// TIA Portal project "DALU-Projekt_HMI_V19" (V19)

(* hardware
DEVICE "SIMATIC 1200-Station_3"  S71200.Device
   slot 0: "S7-1200 Baugruppenträger"  Rack  V1.0
   slot 1: "Target_3"  CPU 1214C DC/DC/DC  6ES7 214-1AE30-0XB0  V2.2
   slot 101: "Target 3 CM 1243-2"  CM 1243-2  3RK7243-2AA30-0XB0  V1.0
   slot 102: "Target 3 CM 1243-5"  CM 1243-5  6GK7 243-5DX30-0XE0  V1.0
DEVICE "ASi-3-S9 (4DI)"  AS-i slave
   slot 0: "-"  Rail
   slot 1: "ASi-3-S9 (4DI)"  AS-i Standard Slave  AS-i Standard Slave Universal
      slot 1: "ASi-3-S9 (4DI) [AS-i Slave (D)]"  AS-i Address-Module
      slot 2: "ASi-3-S9 (4DI) [AS-i Slave (A)]"  AS-i Address-Module
      slot 3: "ASi-3-S9 (4DI) [AS-i Slave (T)]"  AS-i Address-Module
DEVICE "ASi-3-S5 (2AI)"  AS-i slave
   slot 0: "-"  Rail
   slot 1: "ASi-3-S5 (2AI)"  AS-i K60, 2AI-C  3RK1 207-1BQ40-0AA3
      slot 1: "ASi-3-S5 (2AI) [AS-i Slave (D)]"  AS-i Address-Module
      slot 2: "ASi-3-S5 (2AI) [AS-i Slave (A)]"  AS-i Address-Module
      slot 3: "ASi-3-S5 (2AI) [AS-i Slave (T)]"  AS-i Address-Module
DEVICE "ASi-3-S1 (4DI/4DO)"  AS-i slave
   slot 0: "-"  Rail
   slot 1: "ASi-3-S1 (4DI/4DO)"  AS-i 3SB3, 4DI/4DO  3SF5 500-0BC
      slot 1: "ASi-3-S1 (4DI/4DO) [AS-i Slave (D)]"  AS-i Address-Module
      slot 2: "ASi-3-S1 (4DI/4DO) [AS-i Slave (A)]"  AS-i Address-Module
      slot 3: "ASi-3-S1 (4DI/4DO) [AS-i Slave (T)]"  AS-i Address-Module
DEVICE "ASi-3-S7 (2DI,2PO)"  AS-i slave
   slot 0: "-"  Rail
   slot 1: "ASi-3-S7 (2DI,2PO)"  AS-i Standard Slave  AS-i Standard Slave Universal
      slot 1: "ASi-3-S7 (2DI,2PO) [AS-i Slave (D)]"  AS-i Address-Module
      slot 2: "ASi-3-S7 (2DI,2PO) [AS-i Slave (A)]"  AS-i Address-Module
      slot 3: "ASi-3-S7 (2DI,2PO) [AS-i Slave (T)]"  AS-i Address-Module
DEVICE "ASi-3-S3 (2AI)"  AS-i slave
   slot 0: "-"  Rail
   slot 1: "ASi-3-S3 (2AI)"  AS-i K60, 2AI-V  3RK1 207-2BQ40-0AA3
      slot 1: "ASi-3-S3 (2AI) [AS-i Slave (D)]"  AS-i Address-Module
      slot 2: "ASi-3-S3 (2AI) [AS-i Slave (A)]"  AS-i Address-Module
      slot 3: "ASi-3-S3 (2AI) [AS-i Slave (T)]"  AS-i Address-Module
DEVICE "ASi-3-S8 (3DI/1DO)"  AS-i slave
   slot 0: "-"  Rail
   slot 1: "ASi-3-S8 (3DI/1DO)"  AS-i Standard Slave  AS-i Standard Slave Universal
      slot 1: "ASi-3-S8 (3DI/1DO) [AS-i Slave (D)]"  AS-i Address-Module
      slot 2: "ASi-3-S8 (3DI/1DO) [AS-i Slave (A)]"  AS-i Address-Module
      slot 3: "ASi-3-S8 (3DI/1DO) [AS-i Slave (T)]"  AS-i Address-Module
DEVICE "DP_3_S1"  GSD.Device
   slot 0: "Baugruppenträger"  Rail
   slot 0: "DP_3_Simodrive"  6FX2001-5xPxx  4.2
DEVICE "ASi-3-S2 (2AO)"  AS-i slave
   slot 0: "-"  Rail
   slot 1: "ASi-3-S2 (2AO)"  AS-i K60, 2AO-V  3RK1 107-2BQ40-0AA3
      slot 1: "ASi-3-S2 (2AO) [AS-i Slave (D)]"  AS-i Address-Module
      slot 2: "ASi-3-S2 (2AO) [AS-i Slave (A)]"  AS-i Address-Module
      slot 3: "ASi-3-S2 (2AO) [AS-i Slave (T)]"  AS-i Address-Module
DEVICE "ASi-3-S4 (4DI/4DO)"  AS-i slave
   slot 0: "-"  Rail
   slot 1: "ASi-3-S4 (4DI/4DO)"  AS-i K60, 4DI/4DO  3RK1 400-1DQ01-0AA3
      slot 1: "ASi-3-S4 (4DI/4DO) [AS-i Slave (D)]"  AS-i Address-Module
      slot 2: "ASi-3-S4 (4DI/4DO) [AS-i Slave (A)]"  AS-i Address-Module
      slot 3: "ASi-3-S4 (4DI/4DO) [AS-i Slave (T)]"  AS-i Address-Module
DEVICE "ASi-3-S6 (4DI)"  AS-i slave
   slot 0: "-"  Rail
   slot 1: "ASi-3-S6 (4DI)"  AS-i K45, 4DI  3RK1 200-0CQ20-0AA3
      slot 1: "ASi-3-S6 (4DI) [AS-i Slave (D)]"  AS-i Address-Module
      slot 2: "ASi-3-S6 (4DI) [AS-i Slave (A)]"  AS-i Address-Module
      slot 3: "ASi-3-S6 (4DI) [AS-i Slave (T)]"  AS-i Address-Module
DEVICE "SIMATIC 1200-Station_4"  S71200.Device
   slot 0: "S7-1200 Baugruppenträger"  Rack  V1.0
   slot 1: "Target_4"  CPU 1214C DC/DC/DC  6ES7 214-1AE30-0XB0  V2.2
   slot 101: "Target 4 CM 1243-2"  CM 1243-2  3RK7243-2AA30-0XB0  V1.0
   slot 102: "Target 4 CM 1243-5"  CM 1243-5  6GK7 243-5DX30-0XE0  V1.0
DEVICE "ASi-4-S9 (4DI)"  AS-i slave
   slot 0: "-"  Rail
   slot 1: "ASi-4-S9 (4DI)"  AS-i Standard Slave  AS-i Standard Slave Universal
      slot 1: "ASi-4-S9 (4DI) [AS-i Slave (D)]"  AS-i Address-Module
      slot 2: "ASi-4-S9 (4DI) [AS-i Slave (A)]"  AS-i Address-Module
      slot 3: "ASi-4-S9 (4DI) [AS-i Slave (T)]"  AS-i Address-Module
DEVICE "ASi-4-S5 (2AI)"  AS-i slave
   slot 0: "-"  Rail
   slot 1: "ASi-4-S5 (2AI)"  AS-i K60, 2AI-C  3RK1 207-1BQ40-0AA3
      slot 1: "ASi-4-S5 (2AI) [AS-i Slave (D)]"  AS-i Address-Module
      slot 2: "ASi-4-S5 (2AI) [AS-i Slave (A)]"  AS-i Address-Module
      slot 3: "ASi-4-S5 (2AI) [AS-i Slave (T)]"  AS-i Address-Module
DEVICE "ASi-4-S1 (4DI/4DO)"  AS-i slave
   slot 0: "-"  Rail
   slot 1: "ASi-4-S1 (4DI/4DO)"  AS-i 3SB3, 4DI/4DO  3SF5 500-0BC
      slot 1: "ASi-4-S1 (4DI/4DO) [AS-i Slave (D)]"  AS-i Address-Module
      slot 2: "ASi-4-S1 (4DI/4DO) [AS-i Slave (A)]"  AS-i Address-Module
      slot 3: "ASi-4-S1 (4DI/4DO) [AS-i Slave (T)]"  AS-i Address-Module
DEVICE "ASi-4-S7 (2DI,2PO)"  AS-i slave
   slot 0: "-"  Rail
   slot 1: "ASi-4-S7 (2DI,2PO)"  AS-i Standard Slave  AS-i Standard Slave Universal
      slot 1: "ASi-4-S7 (2DI,2PO) [AS-i Slave (D)]"  AS-i Address-Module
      slot 2: "ASi-4-S7 (2DI,2PO) [AS-i Slave (A)]"  AS-i Address-Module
      slot 3: "ASi-4-S7 (2DI,2PO) [AS-i Slave (T)]"  AS-i Address-Module
DEVICE "ASi-4-S3 (2AI)"  AS-i slave
   slot 0: "-"  Rail
   slot 1: "ASi-4-S3 (2AI)"  AS-i K60, 2AI-V  3RK1 207-2BQ40-0AA3
      slot 1: "ASi-4-S3 (2AI) [AS-i Slave (D)]"  AS-i Address-Module
      slot 2: "ASi-4-S3 (2AI) [AS-i Slave (A)]"  AS-i Address-Module
      slot 3: "ASi-4-S3 (2AI) [AS-i Slave (T)]"  AS-i Address-Module
DEVICE "ASi-4-S8 (3DI/1DO)"  AS-i slave
   slot 0: "-"  Rail
   slot 1: "ASi-4-S8 (3DI/1DO)"  AS-i Standard Slave  AS-i Standard Slave Universal
      slot 1: "ASi-4-S8 (3DI/1DO) [AS-i Slave (D)]"  AS-i Address-Module
      slot 2: "ASi-4-S8 (3DI/1DO) [AS-i Slave (A)]"  AS-i Address-Module
      slot 3: "ASi-4-S8 (3DI/1DO) [AS-i Slave (T)]"  AS-i Address-Module
DEVICE "DP_4_S1"  GSD.Device
   slot 0: "Baugruppenträger"  Rail
   slot 0: "DP_4_Simodrive"  6FX2001-5xPxx  4.2
DEVICE "ASi-4-S2 (2AO)"  AS-i slave
   slot 0: "-"  Rail
   slot 1: "ASi-4-S2 (2AO)"  AS-i K60, 2AO-V  3RK1 107-2BQ40-0AA3
      slot 1: "ASi-4-S2 (2AO) [AS-i Slave (D)]"  AS-i Address-Module
      slot 2: "ASi-4-S2 (2AO) [AS-i Slave (A)]"  AS-i Address-Module
      slot 3: "ASi-4-S2 (2AO) [AS-i Slave (T)]"  AS-i Address-Module
DEVICE "ASi-4-S4 (4DI/4DO)"  AS-i slave
   slot 0: "-"  Rail
   slot 1: "ASi-4-S4 (4DI/4DO)"  AS-i K60, 4DI/4DO  3RK1 400-1DQ01-0AA3
      slot 1: "ASi-4-S4 (4DI/4DO) [AS-i Slave (D)]"  AS-i Address-Module
      slot 2: "ASi-4-S4 (4DI/4DO) [AS-i Slave (A)]"  AS-i Address-Module
      slot 3: "ASi-4-S4 (4DI/4DO) [AS-i Slave (T)]"  AS-i Address-Module
DEVICE "ASi-4-S6 (4DI)"  AS-i slave
   slot 0: "-"  Rail
   slot 1: "ASi-4-S6 (4DI)"  AS-i K45, 4DI  3RK1 200-0CQ20-0AA3
      slot 1: "ASi-4-S6 (4DI) [AS-i Slave (D)]"  AS-i Address-Module
      slot 2: "ASi-4-S6 (4DI) [AS-i Slave (A)]"  AS-i Address-Module
      slot 3: "ASi-4-S6 (4DI) [AS-i Slave (T)]"  AS-i Address-Module
DEVICE "SIMATIC 1200-Station_5"  S71200.Device
   slot 0: "S7-1200 Baugruppenträger"  Rack  V1.0
   slot 1: "Target_5"  CPU 1214C DC/DC/DC  6ES7 214-1AE30-0XB0  V2.2
   slot 101: "Target 5 CM 1243-2"  CM 1243-2  3RK7243-2AA30-0XB0  V1.0
   slot 102: "Target 5 CM 1243-5"  CM 1243-5  6GK7 243-5DX30-0XE0  V1.0
DEVICE "ASi-5-S9 (4DI)"  AS-i slave
   slot 0: "-"  Rail
   slot 1: "ASi-5-S9 (4DI)"  AS-i Standard Slave  AS-i Standard Slave Universal
      slot 1: "ASi-5-S9 (4DI) [AS-i Slave (D)]"  AS-i Address-Module
      slot 2: "ASi-5-S9 (4DI) [AS-i Slave (A)]"  AS-i Address-Module
      slot 3: "ASi-5-S9 (4DI) [AS-i Slave (T)]"  AS-i Address-Module
DEVICE "ASi-5-S5 (2AI)"  AS-i slave
   slot 0: "-"  Rail
   slot 1: "ASi-5-S5 (2AI)"  AS-i K60, 2AI-C  3RK1 207-1BQ40-0AA3
      slot 1: "ASi-5-S5 (2AI) [AS-i Slave (D)]"  AS-i Address-Module
      slot 2: "ASi-5-S5 (2AI) [AS-i Slave (A)]"  AS-i Address-Module
      slot 3: "ASi-5-S5 (2AI) [AS-i Slave (T)]"  AS-i Address-Module
DEVICE "ASi-5-S3 (2AI)"  AS-i slave
   slot 0: "-"  Rail
   slot 1: "ASi-5-S3 (2AI)"  AS-i K60, 2AI-V  3RK1 207-2BQ40-0AA3
      slot 1: "ASi-5-S3 (2AI) [AS-i Slave (D)]"  AS-i Address-Module
      slot 2: "ASi-5-S3 (2AI) [AS-i Slave (A)]"  AS-i Address-Module
      slot 3: "ASi-5-S3 (2AI) [AS-i Slave (T)]"  AS-i Address-Module
DEVICE "ASi-5-S7 (2DI,2PO)"  AS-i slave
   slot 0: "-"  Rail
   slot 1: "ASi-5-S7 (2DI,2PO)"  AS-i Standard Slave  AS-i Standard Slave Universal
      slot 1: "ASi-5-S7 (2DI,2PO) [AS-i Slave (D)]"  AS-i Address-Module
      slot 2: "ASi-5-S7 (2DI,2PO) [AS-i Slave (A)]"  AS-i Address-Module
      slot 3: "ASi-5-S7 (2DI,2PO) [AS-i Slave (T)]"  AS-i Address-Module
DEVICE "ASi-5-S2 (2AO)"  AS-i slave
   slot 0: "-"  Rail
   slot 1: "ASi-5-S2 (2AO)"  AS-i K60, 2AO-V  3RK1 107-2BQ40-0AA3
      slot 1: "ASi-5-S2 (2AO) [AS-i Slave (D)]"  AS-i Address-Module
      slot 2: "ASi-5-S2 (2AO) [AS-i Slave (A)]"  AS-i Address-Module
      slot 3: "ASi-5-S2 (2AO) [AS-i Slave (T)]"  AS-i Address-Module
DEVICE "ASi-5-S8 (3DI/1DO)"  AS-i slave
   slot 0: "-"  Rail
   slot 1: "ASi-5-S8 (3DI/1DO)"  AS-i Standard Slave  AS-i Standard Slave Universal
      slot 1: "ASi-5-S8 (3DI/1DO) [AS-i Slave (D)]"  AS-i Address-Module
      slot 2: "ASi-5-S8 (3DI/1DO) [AS-i Slave (A)]"  AS-i Address-Module
      slot 3: "ASi-5-S8 (3DI/1DO) [AS-i Slave (T)]"  AS-i Address-Module
DEVICE "ASi-5-S1 (4DI/4DO)"  AS-i slave
   slot 0: "-"  Rail
   slot 1: "ASi-5-S1 (4DI/4DO)"  AS-i 3SB3, 4DI/4DO  3SF5 500-0BC
      slot 1: "ASi-5-S1 (4DI/4DO) [AS-i Slave (D)]"  AS-i Address-Module
      slot 2: "ASi-5-S1 (4DI/4DO) [AS-i Slave (A)]"  AS-i Address-Module
      slot 3: "ASi-5-S1 (4DI/4DO) [AS-i Slave (T)]"  AS-i Address-Module
DEVICE "DP_5_S1"  GSD.Device
   slot 0: "Baugruppenträger"  Rail
   slot 0: "DP_5_Simodrive"  6FX2001-5xPxx  4.2
DEVICE "ASi-5-S4 (4DI/4DO)"  AS-i slave
   slot 0: "-"  Rail
   slot 1: "ASi-5-S4 (4DI/4DO)"  AS-i K60, 4DI/4DO  3RK1 400-1DQ01-0AA3
      slot 1: "ASi-5-S4 (4DI/4DO) [AS-i Slave (D)]"  AS-i Address-Module
      slot 2: "ASi-5-S4 (4DI/4DO) [AS-i Slave (A)]"  AS-i Address-Module
      slot 3: "ASi-5-S4 (4DI/4DO) [AS-i Slave (T)]"  AS-i Address-Module
DEVICE "ASi-5-S6 (4DI)"  AS-i slave
   slot 0: "-"  Rail
   slot 1: "ASi-5-S6 (4DI)"  AS-i K45, 4DI  3RK1 200-0CQ20-0AA3
      slot 1: "ASi-5-S6 (4DI) [AS-i Slave (D)]"  AS-i Address-Module
      slot 2: "ASi-5-S6 (4DI) [AS-i Slave (A)]"  AS-i Address-Module
      slot 3: "ASi-5-S6 (4DI) [AS-i Slave (T)]"  AS-i Address-Module
DEVICE "SIMATIC 1200-Station_1"  S71200.Device
   slot 0: "S7-1200 Baugruppenträger"  Rack  V1.0
   slot 1: "Target_1"  CPU 1214C DC/DC/DC  6ES7 214-1AE30-0XB0  V2.2
   slot 101: "Target 1 CM 1243-2"  CM 1243-2  3RK7243-2AA30-0XB0  V1.0
   slot 102: "Target 1 CM 1243-5"  CM 1243-5  6GK7 243-5DX30-0XE0  V1.0
DEVICE "ASi-1-S1 (4DI/4DO)"  AS-i slave
   slot 0: "-"  Rail
   slot 1: "ASi-1-S1 (4DI/4DO)"  AS-i 3SB3, 4DI/4DO  3SF5 500-0BC
      slot 1: "ASi-1-S1 (4DI/4DO) [AS-i Slave (D)]"  AS-i Address-Module
      slot 2: "ASi-1-S1 (4DI/4DO) [AS-i Slave (A)]"  AS-i Address-Module
      slot 3: "ASi-1-S1 (4DI/4DO) [AS-i Slave (T)]"  AS-i Address-Module
DEVICE "DP_1_S1"  GSD.Device
   slot 0: "Baugruppenträger"  Rail
   slot 0: "DP_1_Simodrive"  6FX2001-5xPxx  4.2
DEVICE "ASi-1-S4 (4DI/4DO)"  AS-i slave
   slot 0: "-"  Rail
   slot 1: "ASi-1-S4 (4DI/4DO)"  AS-i K60, 4DI/4DO  3RK1 400-1DQ01-0AA3
      slot 1: "ASi-1-S4 (4DI/4DO) [AS-i Slave (D)]"  AS-i Address-Module
      slot 2: "ASi-1-S4 (4DI/4DO) [AS-i Slave (A)]"  AS-i Address-Module
      slot 3: "ASi-1-S4 (4DI/4DO) [AS-i Slave (T)]"  AS-i Address-Module
DEVICE "ASi-1-S6 (4DI)"  AS-i slave
   slot 0: "-"  Rail
   slot 1: "ASi-1-S6 (4DI)"  AS-i K45, 4DI  3RK1 200-0CQ20-0AA3
      slot 1: "ASi-1-S6 (4DI) [AS-i Slave (D)]"  AS-i Address-Module
      slot 2: "ASi-1-S6 (4DI) [AS-i Slave (A)]"  AS-i Address-Module
      slot 3: "ASi-1-S6 (4DI) [AS-i Slave (T)]"  AS-i Address-Module
DEVICE "ASi-1-S9 (4DI)"  AS-i slave
   slot 0: "-"  Rail
   slot 1: "ASi-1-S9 (4DI)"  AS-i Standard Slave  AS-i Standard Slave Universal
      slot 1: "ASi-1-S9 (4DI) [AS-i Slave (D)]"  AS-i Address-Module
      slot 2: "ASi-1-S9 (4DI) [AS-i Slave (A)]"  AS-i Address-Module
      slot 3: "ASi-1-S9 (4DI) [AS-i Slave (T)]"  AS-i Address-Module
DEVICE "ASi-1-S5 (2AI)"  AS-i slave
   slot 0: "-"  Rail
   slot 1: "ASi-1-S5 (2AI)"  AS-i K60, 2AI-C  3RK1 207-1BQ40-0AA3
      slot 1: "ASi-1-S5 (2AI) [AS-i Slave (D)]"  AS-i Address-Module
      slot 2: "ASi-1-S5 (2AI) [AS-i Slave (A)]"  AS-i Address-Module
      slot 3: "ASi-1-S5 (2AI) [AS-i Slave (T)]"  AS-i Address-Module
DEVICE "ASi-1-S3 (2AI)"  AS-i slave
   slot 0: "-"  Rail
   slot 1: "ASi-1-S3 (2AI)"  AS-i K60, 2AI-V  3RK1 207-2BQ40-0AA3
      slot 1: "ASi-1-S3 (2AI) [AS-i Slave (D)]"  AS-i Address-Module
      slot 2: "ASi-1-S3 (2AI) [AS-i Slave (A)]"  AS-i Address-Module
      slot 3: "ASi-1-S3 (2AI) [AS-i Slave (T)]"  AS-i Address-Module
DEVICE "ASi-1-S7 (2DI,2PO)"  AS-i slave
   slot 0: "-"  Rail
   slot 1: "ASi-1-S7 (2DI,2PO)"  AS-i Standard Slave  AS-i Standard Slave Universal
      slot 1: "ASi-1-S7 (2DI,2PO) [AS-i Slave (D)]"  AS-i Address-Module
      slot 2: "ASi-1-S7 (2DI,2PO) [AS-i Slave (A)]"  AS-i Address-Module
      slot 3: "ASi-1-S7 (2DI,2PO) [AS-i Slave (T)]"  AS-i Address-Module
DEVICE "ASi-1-S2 (2AO)"  AS-i slave
   slot 0: "-"  Rail
   slot 1: "ASi-1-S2 (2AO)"  AS-i K60, 2AO-V  3RK1 107-2BQ40-0AA3
      slot 1: "ASi-1-S2 (2AO) [AS-i Slave (D)]"  AS-i Address-Module
      slot 2: "ASi-1-S2 (2AO) [AS-i Slave (A)]"  AS-i Address-Module
      slot 3: "ASi-1-S2 (2AO) [AS-i Slave (T)]"  AS-i Address-Module
DEVICE "ASi-1-S8 (3DI/1DO)"  AS-i slave
   slot 0: "-"  Rail
   slot 1: "ASi-1-S8 (3DI/1DO)"  AS-i Standard Slave  AS-i Standard Slave Universal
      slot 1: "ASi-1-S8 (3DI/1DO) [AS-i Slave (D)]"  AS-i Address-Module
      slot 2: "ASi-1-S8 (3DI/1DO) [AS-i Slave (A)]"  AS-i Address-Module
      slot 3: "ASi-1-S8 (3DI/1DO) [AS-i Slave (T)]"  AS-i Address-Module
DEVICE "ASi-2-S8 (3DI/1DO)"  AS-i slave
   slot 0: "-"  Rail
   slot 1: "ASi-2-S8 (3DI/1DO)"  AS-i Standard Slave  AS-i Standard Slave Universal
      slot 1: "ASi-2-S8 (3DI/1DO) [AS-i Slave (D)]"  AS-i Address-Module
      slot 2: "ASi-2-S8 (3DI/1DO) [AS-i Slave (A)]"  AS-i Address-Module
      slot 3: "ASi-2-S8 (3DI/1DO) [AS-i Slave (T)]"  AS-i Address-Module
DEVICE "ASi-2-S2 (2AO)"  AS-i slave
   slot 0: "-"  Rail
   slot 1: "ASi-2-S2 (2AO)"  AS-i K60, 2AO-V  3RK1 107-2BQ40-0AA3
      slot 1: "ASi-2-S2 (2AO) [AS-i Slave (D)]"  AS-i Address-Module
      slot 2: "ASi-2-S2 (2AO) [AS-i Slave (A)]"  AS-i Address-Module
      slot 3: "ASi-2-S2 (2AO) [AS-i Slave (T)]"  AS-i Address-Module
DEVICE "ASi-2-S7 (2DI,2PO)"  AS-i slave
   slot 0: "-"  Rail
   slot 1: "ASi-2-S7 (2DI,2PO)"  AS-i Standard Slave  AS-i Standard Slave Universal
      slot 1: "ASi-2-S7 (2DI,2PO) [AS-i Slave (D)]"  AS-i Address-Module
      slot 2: "ASi-2-S7 (2DI,2PO) [AS-i Slave (A)]"  AS-i Address-Module
      slot 3: "ASi-2-S7 (2DI,2PO) [AS-i Slave (T)]"  AS-i Address-Module
DEVICE "ASi-2-S3 (2AI)"  AS-i slave
   slot 0: "-"  Rail
   slot 1: "ASi-2-S3 (2AI)"  AS-i K60, 2AI-V  3RK1 207-2BQ40-0AA3
      slot 1: "ASi-2-S3 (2AI) [AS-i Slave (D)]"  AS-i Address-Module
      slot 2: "ASi-2-S3 (2AI) [AS-i Slave (A)]"  AS-i Address-Module
      slot 3: "ASi-2-S3 (2AI) [AS-i Slave (T)]"  AS-i Address-Module
DEVICE "ASi-2-S5 (2AI)"  AS-i slave
   slot 0: "-"  Rail
   slot 1: "ASi-2-S5 (2AI)"  AS-i K60, 2AI-C  3RK1 207-1BQ40-0AA3
      slot 1: "ASi-2-S5 (2AI) [AS-i Slave (D)]"  AS-i Address-Module
      slot 2: "ASi-2-S5 (2AI) [AS-i Slave (A)]"  AS-i Address-Module
      slot 3: "ASi-2-S5 (2AI) [AS-i Slave (T)]"  AS-i Address-Module
DEVICE "ASi-2-S9 (4DI)"  AS-i slave
   slot 0: "-"  Rail
   slot 1: "ASi-2-S9 (4DI)"  AS-i Standard Slave  AS-i Standard Slave Universal
      slot 1: "ASi-2-S9 (4DI) [AS-i Slave (D)]"  AS-i Address-Module
      slot 2: "ASi-2-S9 (4DI) [AS-i Slave (A)]"  AS-i Address-Module
      slot 3: "ASi-2-S9 (4DI) [AS-i Slave (T)]"  AS-i Address-Module
DEVICE "ASi-2-S4 (4DI/4DO)"  AS-i slave
   slot 0: "-"  Rail
   slot 1: "ASi-2-S4 (4DI/4DO)"  AS-i K60, 4DI/4DO  3RK1 400-1DQ01-0AA3
      slot 1: "ASi-2-S4 (4DI/4DO) [AS-i Slave (D)]"  AS-i Address-Module
      slot 2: "ASi-2-S4 (4DI/4DO) [AS-i Slave (A)]"  AS-i Address-Module
      slot 3: "ASi-2-S4 (4DI/4DO) [AS-i Slave (T)]"  AS-i Address-Module
DEVICE "DP_2_S1"  GSD.Device
   slot 0: "Baugruppenträger"  Rail
   slot 0: "DP_2_Simodrive"  6FX2001-5xPxx  4.2
DEVICE "ASi-2-S1 (4DI/4DO)"  AS-i slave
   slot 0: "-"  Rail
   slot 1: "ASi-2-S1 (4DI/4DO)"  AS-i 3SB3, 4DI/4DO  3SF5 500-0BC
      slot 1: "ASi-2-S1 (4DI/4DO) [AS-i Slave (D)]"  AS-i Address-Module
      slot 2: "ASi-2-S1 (4DI/4DO) [AS-i Slave (A)]"  AS-i Address-Module
      slot 3: "ASi-2-S1 (4DI/4DO) [AS-i Slave (T)]"  AS-i Address-Module
DEVICE "SIMATIC 1200-Station_2"  S71200.Device
   slot 0: "S7-1200 Baugruppenträger"  Rack  V1.0
   slot 1: "Target_2"  CPU 1214C DC/DC/DC  6ES7 214-1AE30-0XB0  V2.2
   slot 101: "Target 2 CM 1243-2"  CM 1243-2  3RK7243-2AA30-0XB0  V1.0
   slot 102: "Target 2 CM 1243-5"  CM 1243-5  6GK7 243-5DX30-0XE0  V1.0
DEVICE "ASi-2-S6 (4DI)"  AS-i slave
   slot 0: "-"  Rail
   slot 1: "ASi-2-S6 (4DI)"  AS-i K45, 4DI, A/B  3RK2 200-0CQ20-0AA3
      slot 1: "ASi-2-S6 (4DI) [AS-i Slave (D)]"  AS-i Address-Module
      slot 2: "ASi-2-S6 (4DI) [AS-i Slave (A)]"  AS-i Address-Module
      slot 3: "ASi-2-S6 (4DI) [AS-i Slave (T)]"  AS-i Address-Module
DEVICE "HMI_1"  KTP400 Comfort
   slot 0: "HMI_1"  KTP400 Comfort  6AV2 124-2DC01-0AX0  15.1.0.0
   slot 1: "HMI_RT_1"  KTP400 Comfort  6AV2 124-2DC01-0AX0  15.1.0.0
   slot 5: "HMI_1.IE_CP_1"  PROFINET Interface  15.0.1.0
      slot 1: "PROFINET Interface_1"  PROFINET Interface
         slot 1: "Port_1"  Port
   slot 7: "HMI_1.MPI/DP_CP_1"  MPI/DP Interface  15.0.1.0
DEVICE "HMI_2"  KTP400 Comfort
   slot 0: "HMI_1"  KTP400 Comfort  6AV2 124-2DC01-0AX0  15.1.0.0
   slot 1: "HMI_RT_2"  KTP400 Comfort  6AV2 124-2DC01-0AX0  15.1.0.0
   slot 5: "HMI_1.IE_CP_1"  PROFINET Interface  15.0.1.0
      slot 1: "PROFINET Interface_1"  PROFINET Interface
         slot 1: "Port_1"  Port
   slot 7: "HMI_1.MPI/DP_CP_1"  MPI/DP Interface  15.0.1.0
DEVICE "HMI_3"  KTP400 Comfort
   slot 0: "HMI_1"  KTP400 Comfort  6AV2 124-2DC01-0AX0  15.1.0.0
   slot 1: "HMI_RT_3"  KTP400 Comfort  6AV2 124-2DC01-0AX0  15.1.0.0
   slot 5: "HMI_1.IE_CP_1"  PROFINET Interface  15.0.1.0
      slot 1: "PROFINET Interface_1"  PROFINET Interface
         slot 1: "Port_1"  Port
   slot 7: "HMI_1.MPI/DP_CP_1"  MPI/DP Interface  15.0.1.0
DEVICE "HMI_4"  KTP400 Comfort
   slot 0: "HMI_1"  KTP400 Comfort  6AV2 124-2DC01-0AX0  15.1.0.0
   slot 1: "HMI_RT_4"  KTP400 Comfort  6AV2 124-2DC01-0AX0  15.1.0.0
   slot 5: "HMI_1.IE_CP_1"  PROFINET Interface  15.0.1.0
      slot 1: "PROFINET Interface_1"  PROFINET Interface
         slot 1: "Port_1"  Port
   slot 7: "HMI_1.MPI/DP_CP_1"  MPI/DP Interface  15.0.1.0
DEVICE "HMI_5"  KTP400 Comfort
   slot 0: "HMI_1"  KTP400 Comfort  6AV2 124-2DC01-0AX0  15.1.0.0
   slot 1: "HMI_RT_5"  KTP400 Comfort  6AV2 124-2DC01-0AX0  15.1.0.0
   slot 5: "HMI_1.IE_CP_1"  PROFINET Interface  15.0.1.0
      slot 1: "PROFINET Interface_1"  PROFINET Interface
         slot 1: "Port_1"  Port
   slot 7: "HMI_1.MPI/DP_CP_1"  MPI/DP Interface  15.0.1.0
*)

// ===== PLC "Target_3"  CPU 1214C DC/DC/DC =====

VAR_GLOBAL   // PLC tag table "Standard-Variablentabelle"
   "Clock_2.5Hz" AT %M8000.2 : Bool;
   "Clock_2Hz" AT %M8000.3 : Bool;
   "Clock_1.25Hz" AT %M8000.4 : Bool;
   "Clock_1Hz" AT %M8000.5 : Bool;
   "Clock_0.625Hz" AT %M8000.6 : Bool;
   "Clock_0.5Hz" AT %M8000.7 : Bool;
   "System_Byte" AT %MB8001 : Byte;
   "FirstScan" AT %M8001.0 : Bool;
   "AlwaysTRUE" AT %M8001.2 : Bool;
   "AlwaysFALSE" AT %M8001.3 : Bool;
   "LAMPE_0" AT %Q2.0 : Bool;
   "TAST_0" AT %I2.0 : Bool;
   "MAGE_U" AT %I7.1 : Bool;
   "MAGE_D" AT %I7.2 : Bool;
   "MCGo" AT %Q5.2 : Bool;
   "MCDir" AT %Q5.3 : Bool;
   "LAMPE_1" AT %Q2.1 : Bool;
   "LAMPE_2" AT %Q2.2 : Bool;
   "LAMPE_3" AT %Q2.3 : Bool;
   "TAST_1" AT %I2.1 : Bool;
   "GlasLS" AT %I7.0 : Bool;
   "KapNS" AT %I5.2 : Bool;
   "OptNS" AT %I5.3 : Bool;
   "IndNS_0" AT %I9.0 : Bool;
   "IndNS_1" AT %I9.1 : Bool;
   "IndNS_2" AT %I9.2 : Bool;
   "SONAR" AT %I10.0 : Bool;
   "EinLS" AT %I5.0 : Bool;
   "LED0" AT %Q0.0 : Bool;
   "LED1" AT %Q0.1 : Bool;
   "LED2" AT %Q0.2 : Bool;
   "LED3" AT %Q0.3 : Bool;
   "LED4" AT %Q0.4 : Bool;
   "LED5" AT %Q0.5 : Bool;
   "LED6" AT %Q0.6 : Bool;
   "LED7" AT %Q0.7 : Bool;
   "PosElM" AT %I1.0 : Bool;
END_VAR

DATA_BLOCK "DB"   // DB1
{ S7_Optimized_Access := 'TRUE' }
VERSION : 0.1
   VAR
      motor_state : Byte;
   END_VAR
BEGIN
END_DATA_BLOCK

ORGANIZATION_BLOCK "main"   // OB1, SCL, ProgramCycle
TITLE = "Main Program Sweep (Cycle)"
{ S7_Optimized_Access := 'TRUE' }
VERSION : 0.1
   VAR CONSTANT
      motor_reset : Byte;
      motor_down : Byte := 16#1;
      motor_up : Byte := 16#2;
   END_VAR
BEGIN
   "LED0" := "GlasLS";
   "LED1" := "KapNS";
   "LED2" := "OptNS";
   "LED3" := "SONAR";
   "LED4" := "EinLS";
   "LED5" := "IndNS_0";
   "LED6" := "IndNS_1";
   "LED7" := "PosElM";
END_ORGANIZATION_BLOCK

// ===== PLC "Target_4"  CPU 1214C DC/DC/DC =====

VAR_GLOBAL   // PLC tag table "Standard-Variablentabelle"
   "Clock_2.5Hz" AT %M8000.2 : Bool;
   "Clock_2Hz" AT %M8000.3 : Bool;
   "Clock_1.25Hz" AT %M8000.4 : Bool;
   "Clock_1Hz" AT %M8000.5 : Bool;
   "Clock_0.625Hz" AT %M8000.6 : Bool;
   "Clock_0.5Hz" AT %M8000.7 : Bool;
   "System_Byte" AT %MB8001 : Byte;
   "FirstScan" AT %M8001.0 : Bool;
   "AlwaysTRUE" AT %M8001.2 : Bool;
   "AlwaysFALSE" AT %M8001.3 : Bool;
END_VAR

ORGANIZATION_BLOCK "Main"   // OB1, LAD, ProgramCycle
TITLE = "Main Program Sweep (Cycle)"
{ S7_Optimized_Access := 'TRUE' }
VERSION : 0.1
BEGIN
END_ORGANIZATION_BLOCK

// ===== PLC "Target_5"  CPU 1214C DC/DC/DC =====

VAR_GLOBAL   // PLC tag table "Standard-Variablentabelle"
   "Clock_2.5Hz" AT %M8000.2 : Bool;
   "Clock_2Hz" AT %M8000.3 : Bool;
   "Clock_1.25Hz" AT %M8000.4 : Bool;
   "Clock_1Hz" AT %M8000.5 : Bool;
   "Clock_0.625Hz" AT %M8000.6 : Bool;
   "Clock_0.5Hz" AT %M8000.7 : Bool;
   "System_Byte" AT %MB8001 : Byte;
   "FirstScan" AT %M8001.0 : Bool;
   "AlwaysTRUE" AT %M8001.2 : Bool;
   "AlwaysFALSE" AT %M8001.3 : Bool;
END_VAR

ORGANIZATION_BLOCK "Main"   // OB1, LAD, ProgramCycle
TITLE = "Main Program Sweep (Cycle)"
{ S7_Optimized_Access := 'TRUE' }
VERSION : 0.1
BEGIN
END_ORGANIZATION_BLOCK

// ===== PLC "Target_1"  CPU 1214C DC/DC/DC =====

VAR_GLOBAL   // PLC tag table "Standard-Variablentabelle"
   "Clock_2.5Hz" AT %M8000.2 : Bool;
   "Clock_2Hz" AT %M8000.3 : Bool;
   "Clock_1.25Hz" AT %M8000.4 : Bool;
   "Clock_1Hz" AT %M8000.5 : Bool;
   "Clock_0.625Hz" AT %M8000.6 : Bool;
   "Clock_0.5Hz" AT %M8000.7 : Bool;
   "System_Byte" AT %MB8001 : Byte;
   "FirstScan" AT %M8001.0 : Bool;
   "AlwaysTRUE" AT %M8001.2 : Bool;
   "AlwaysFALSE" AT %M8001.3 : Bool;
END_VAR

ORGANIZATION_BLOCK "Main"   // OB1, LAD, ProgramCycle
TITLE = "Main Program Sweep (Cycle)"
{ S7_Optimized_Access := 'TRUE' }
VERSION : 0.1
BEGIN
END_ORGANIZATION_BLOCK

// ===== PLC "Target_2"  CPU 1214C DC/DC/DC =====

VAR_GLOBAL   // PLC tag table "Standard-Variablentabelle"
   "Clock_2.5Hz" AT %M8000.2 : Bool;
   "Clock_2Hz" AT %M8000.3 : Bool;
   "Clock_1.25Hz" AT %M8000.4 : Bool;
   "Clock_1Hz" AT %M8000.5 : Bool;
   "Clock_0.625Hz" AT %M8000.6 : Bool;
   "Clock_0.5Hz" AT %M8000.7 : Bool;
   "System_Byte" AT %MB8001 : Byte;
   "FirstScan" AT %M8001.0 : Bool;
   "AlwaysTRUE" AT %M8001.2 : Bool;
   "AlwaysFALSE" AT %M8001.3 : Bool;
END_VAR

ORGANIZATION_BLOCK "Main"   // OB1, LAD, ProgramCycle
TITLE = "Main Program Sweep (Cycle)"
{ S7_Optimized_Access := 'TRUE' }
VERSION : 0.1
BEGIN
END_ORGANIZATION_BLOCK

(* ===== HMI "HMI_RT_1" =====
system functions are stored by id; their names below are inferred from use
connection "HMI_Connection_1": ETHERNET, S7_1200_OMS

HMI tags "Default tag table"
   "Tag_ScreenNumber" : UInt, internal

text list "Textliste_Bildnamen": 1 'Root screen'

screen "Root screen" 480x212, template "Template_1"
   on GenerateScreen: SetTag("Tag_ScreenNumber", 1)
   TextField "HmiScreenItemData" at 48,60 size 384x22; Text 'Willkommen zum HMI_1 (KTP400 Comfort)!'

Template "Template_1" 480x212
   Button "Beenden" at 379,148 size 63x63; TextOff 'Beenden'; PictureOff "ExitRuntime_KTP400_Comfort_TR"; PictureOn "ExitRuntime_KTP400_Comfort_TR"
      on Release: StopRuntime(0)
   Button "Template_Button" at 265,148 size 63x63; TextOff 'Text'
   Button "Meldungen" at 151,148 size 63x63; TextOff 'Meldungen'; PictureOff "AlarmDisplay_KTP400_Comfort_TR"; PictureOn "AlarmDisplay_KTP400_Comfort_TR"
      on Release: function_ef3f5d25("Alarm window_Unacknowledged", -1)
   Button "Startbild" at 37,148 size 63x63; TextOff 'Startbild'; PictureOff "NavigateHome_KTP400_Comfort_TR"; PictureOn "NavigateHome_KTP400_Comfort_TR"
      on Release: ActivateScreen("Root screen", 0)
*)

(* ===== HMI "HMI_RT_2" =====
system functions are stored by id; their names below are inferred from use
connection "HMI_Connection_2": ETHERNET, S7_1200_OMS

HMI tags "Default tag table"
   "Tag_ScreenNumber" : UInt, internal

text list "Textliste_Bildnamen": 1 'Root screen'

screen "Root screen" 480x212, template "Template_1"
   on GenerateScreen: SetTag("Tag_ScreenNumber", 1)
   TextField "HmiScreenItemData" at 48,60 size 384x22; Text 'Willkommen zum HMI_2 (KTP400 Comfort)!'

Template "Template_1" 480x212
   Button "Beenden" at 379,148 size 63x63; TextOn 'Beenden'; TextOff 'Beenden'; PictureOn "ExitRuntime_KTP400_Comfort_TR"; PictureOff "ExitRuntime_KTP400_Comfort_TR"
      on Release: StopRuntime(0)
   Button "Template_Button" at 265,148 size 63x63; TextOff 'Text'
   Button "Meldungen" at 151,148 size 63x63; TextOn 'Meldungen'; TextOff 'Meldungen'; PictureOn "AlarmDisplay_KTP400_Comfort_TR"; PictureOff "AlarmDisplay_KTP400_Comfort_TR"
      on Release: function_ef3f5d25("Alarm window_Unacknowledged", -1)
   Button "Startbild" at 37,148 size 63x63; TextOn 'Startbild'; TextOff 'Startbild'; PictureOn "NavigateHome_KTP400_Comfort_TR"; PictureOff "NavigateHome_KTP400_Comfort_TR"
      on Release: ActivateScreen("Root screen", 0)
*)

(* ===== HMI "HMI_RT_3" =====
system functions are stored by id; their names below are inferred from use
connection "HMI_Connection_3": ETHERNET, S7_1200_OMS

HMI tags "Default tag table"
   "Tag_ScreenNumber" : UInt, internal

text list "Textliste_Bildnamen": 1 'Root screen'

screen "Root screen" 480x212, template "Template_1"
   on GenerateScreen: SetTag("Tag_ScreenNumber", 1)
   TextField "HmiScreenItemData" at 48,60 size 384x22; Text 'Willkommen zum HMI_3 (KTP400 Comfort)!'

Template "Template_1" 480x212
   Button "Beenden" at 379,148 size 63x63; TextOn 'Beenden'; TextOff 'Beenden'; PictureOn "ExitRuntime_KTP400_Comfort_TR"; PictureOff "ExitRuntime_KTP400_Comfort_TR"
      on Release: StopRuntime(0)
   Button "Template_Button" at 265,148 size 63x63; TextOff 'Text'
   Button "Meldungen" at 151,148 size 63x63; TextOn 'Meldungen'; TextOff 'Meldungen'; PictureOn "AlarmDisplay_KTP400_Comfort_TR"; PictureOff "AlarmDisplay_KTP400_Comfort_TR"
      on Release: function_ef3f5d25("Alarm window_Unacknowledged", -1)
   Button "Startbild" at 37,148 size 63x63; TextOn 'Startbild'; TextOff 'Startbild'; PictureOn "NavigateHome_KTP400_Comfort_TR"; PictureOff "NavigateHome_KTP400_Comfort_TR"
      on Release: ActivateScreen("Root screen", 0)
*)

(* ===== HMI "HMI_RT_4" =====
system functions are stored by id; their names below are inferred from use
connection "HMI_Connection_4": ETHERNET, S7_1200_OMS

HMI tags "Default tag table"
   "Tag_ScreenNumber" : UInt, internal

text list "Textliste_Bildnamen": 1 'Root screen'

screen "Root screen" 480x212, template "Template_1"
   on GenerateScreen: SetTag("Tag_ScreenNumber", 1)
   TextField "HmiScreenItemData" at 48,60 size 384x22; Text 'Willkommen zum HMI_4 (KTP400 Comfort)!'

Template "Template_1" 480x212
   Button "Beenden" at 379,148 size 63x63; TextOn 'Beenden'; TextOff 'Beenden'; PictureOn "ExitRuntime_KTP400_Comfort_TR"; PictureOff "ExitRuntime_KTP400_Comfort_TR"
      on Release: StopRuntime(0)
   Button "Template_Button" at 265,148 size 63x63; TextOff 'Text'
   Button "Meldungen" at 151,148 size 63x63; TextOn 'Meldungen'; TextOff 'Meldungen'; PictureOn "AlarmDisplay_KTP400_Comfort_TR"; PictureOff "AlarmDisplay_KTP400_Comfort_TR"
      on Release: function_ef3f5d25("Alarm window_Unacknowledged", -1)
   Button "Startbild" at 37,148 size 63x63; TextOn 'Startbild'; TextOff 'Startbild'; PictureOn "NavigateHome_KTP400_Comfort_TR"; PictureOff "NavigateHome_KTP400_Comfort_TR"
      on Release: ActivateScreen("Root screen", 0)
*)

(* ===== HMI "HMI_RT_5" =====
system functions are stored by id; their names below are inferred from use
connection "HMI_Connection_5": ETHERNET, S7_1200_OMS

HMI tags "Default tag table"
   "Tag_ScreenNumber" : UInt, internal

text list "Textliste_Bildnamen": 1 'Root screen'

screen "Root screen" 480x212, template "Template_1"
   on GenerateScreen: SetTag("Tag_ScreenNumber", 1)
   TextField "HmiScreenItemData" at 48,60 size 384x22; Text 'Willkommen zum HMI_5 (KTP400 Comfort)!'

Template "Template_1" 480x212
   Button "Beenden" at 379,148 size 63x63; TextOn 'Beenden'; TextOff 'Beenden'; PictureOn "ExitRuntime_KTP400_Comfort_TR"; PictureOff "ExitRuntime_KTP400_Comfort_TR"
      on Release: StopRuntime(0)
   Button "Template_Button" at 265,148 size 63x63; TextOff 'Text'
   Button "Meldungen" at 151,148 size 63x63; TextOn 'Meldungen'; TextOff 'Meldungen'; PictureOn "AlarmDisplay_KTP400_Comfort_TR"; PictureOff "AlarmDisplay_KTP400_Comfort_TR"
      on Release: function_ef3f5d25("Alarm window_Unacknowledged", -1)
   Button "Startbild" at 37,148 size 63x63; TextOn 'Startbild'; TextOff 'Startbild'; PictureOn "NavigateHome_KTP400_Comfort_TR"; PictureOff "NavigateHome_KTP400_Comfort_TR"
      on Release: ActivateScreen("Root screen", 0)
*)